FUNCTION_BLOCK FieldsToArrowheadEvent (* Transform individual fields to an Arrowhead Event type *)
  (* Standard: 61499-2; Description: Copyright (c) 2019 fortiss GmbH This program and the accompanying materials are made available under the terms of the Eclipse Public License 2.0 which is available at https://www.eclipse.org/legal/epl-2.0/ SPDX-License-Identifier: EPL-2.0 *)
  (* Version 1.0, 2019-10-17, Cabral, fortiss GmbH *)
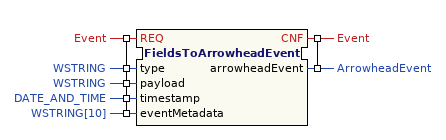
  EVENT_INPUT
    REQ WITH type, payload, timestamp, eventMetadata; (* Normal Execution Request *)
  END_EVENT
  EVENT_OUTPUT
    CNF WITH arrowheadEvent; (* Execution Confirmation *)
  END_EVENT
  VAR_INPUT
    type : WSTRING; (* The type of the event, an event ID of sorts *)
    payload : WSTRING; (* String data of the event *)
    timestamp : DATE_AND_TIME; (* Date and time of the event *)
    eventMetadata : ARRAY [0..9] OF WSTRING; (* Key=value pairs of additional data about the event *)
  END_VAR
  VAR_OUTPUT
    arrowheadEvent : ArrowheadEvent; (* Created Arrowhead event *)
  END_VAR
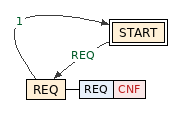
  EC_STATES
    START; (* Initial State *)
    REQ : REQ -> CNF;
  END_STATES
  EC_TRANSITIONS
    REQ TO START := 1;
    START TO REQ := REQ;
  END_TRANSITIONS
  ALGORITHM REQ IN ST: (* Initialization algorithm *)
VAR
  i: INT;
END_VAR;

i := 0;
arrowheadEvent.type := type;
arrowheadEvent.payload := payload;
arrowheadEvent.timestamp = timestamp;

WHILE i < 10 DO //looks like while is faster than FOR when exporting to cpp
  arrowheadEvent.eventMetadata[i] :=  eventMetadata[i];
  i := i + 1;
END_WHILE
  END_ALGORITHM
END_FUNCTION_BLOCK
